DATA_BLOCK "DB_executeQuery2"
{ S7_Optimized_Access := 'TRUE' }
VERSION : 0.1
NON_RETAIN
"FB_ExecuteQuery2"

BEGIN

END_DATA_BLOCK

